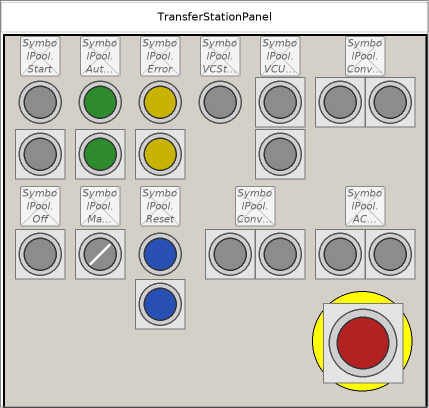
VISUALIZATION V_TransferPanel  // 429x408
VAR_IN_OUT
	Signals : ST_TransferPanel;
END_VAR
    Rectangle (3,34 424x374)
    Ellipse (312,291 100x100)
    PushSwitch (15,129 50x50), tooltip "Activate main contactor", variable: Signals.inputs.PB_ActivateMainContactor, behaviour: TAP, style: Switch-PushSwitch-Gray
    Lamp1 (15,77 50x50), tooltip "Main contactor activeated", variable: Signals.outputs.LED_MainContactorActivated, style: Lamp-Lamp1-Gray
    PushSwitch (75,129 50x50), tooltip "Auto on", variable: Signals.inputs.PB_AutoOn, behaviour: TAP, style: Switch-PushSwitch-Green
    Lamp1 (75,77 50x50), tooltip "Auto activated", variable: Signals.outputs.LED_AutoIsOn, style: Lamp-Lamp1-Green
    Lamp1 (135,77 50x50), tooltip "Error", variable: Signals.outputs.LED_Error, style: Lamp-Lamp1-Yellow
    PushSwitch (135,129 50x50), tooltip "Reset error", variable: Signals.inputs.PB_ErrorReset, behaviour: TAP, style: Switch-PushSwitch-Yellow
    Lamp1 (135,229 50x50), tooltip "Emergency stop", variable: Signals.outputs.LED_EmergencyStop, style: Lamp-Lamp1-Blue
    PushSwitch (135,279 50x50), tooltip "Reset emergency stop", variable: Signals.inputs.PB_EmergencyStopReset, behaviour: TAP, style: Switch-PushSwitch-Blue
    RotarySwitch (75,229 50x50), tooltip "Man/Auto", variable: Signals.inputs.SW_Auto, behaviour: TOGGLE, style: Switch-RotarySwitch-Gray
    Lamp1 (195,77 50x50), tooltip "VC stopped", variable: Signals.outputs.LED_VcStopped, style: Lamp-Lamp1-Gray
    PushSwitch (255,129 50x50), tooltip "VC Down", variable: Signals.inputs.PB_VcDown, behaviour: TAP, style: Switch-PushSwitch-Gray
    PushSwitch (255,77 50x50), tooltip "VC Up", variable: Signals.inputs.PB_VcUp, behaviour: TAP, style: Switch-PushSwitch-Gray
    PushSwitch (365,77 50x50), tooltip "Transfer Conveyor Right", variable: Signals.inputs.PB_Conv_1_Right, behaviour: TAP, style: Switch-PushSwitch-Gray
    PushSwitch (315,77 50x50), tooltip "Transfer Conveyor Left", variable: Signals.inputs.PB_Conv_1_Left, behaviour: TAP, style: Switch-PushSwitch-Gray
    PushSwitch (255,229 50x50), tooltip "VC Conveyor Right", variable: Signals.inputs.PB_VcConvRight, behaviour: TAP, style: Switch-PushSwitch-Gray
    PushSwitch (205,229 50x50), tooltip "VC Conveyor Left", variable: Signals.inputs.PB_VcConvLeft, behaviour: TAP, style: Switch-PushSwitch-Gray
    PushSwitch (365,229 50x50), tooltip "AC Conveyor Right", variable: Signals.inputs.PB_AC_ConvRight, behaviour: TAP, style: Switch-PushSwitch-Gray
    PushSwitch (315,229 50x50), tooltip "AC Conveyor Left", variable: Signals.inputs.PB_AC_ConvLeft, behaviour: TAP, style: Switch-PushSwitch-Gray
    PushSwitch (15,229 50x50), tooltip "Main contactor off", variable: Signals.inputs.PB_MainContactorOff, behaviour: TAP, style: Switch-PushSwitch-Gray
    PushSwitch (323,303 80x80), tooltip "Emergency stop", variable: Signals.inputs.PB_EmergencyStop, behaviour: TOGGLE, style: Switch-PushSwitch-Red
    Image (20,36 40x40), image: SymbolPool.Start
    Image (80,36 40x40), image: SymbolPool.AutoOn
    Image (140,36 40x40), image: SymbolPool.Error
    Image (200,36 40x40), image: SymbolPool.VCStopped
    Image (260,36 40x40), image: SymbolPool.VCUpDown
    Image (345,36 40x40), image: SymbolPool.Conv1_L_R
    Image (235,186 40x40), image: SymbolPool.Conv_L_R
    Image (345,186 40x40), image: SymbolPool.AC_Conv_L_R
    Image (20,186 40x40), image: SymbolPool.Off
    Image (80,186 40x40), image: SymbolPool.ManAuto
    Image (140,186 40x40), image: SymbolPool.Reset
    Textfield (1,2 428x30), "TransferStationPanel"
END_VISUALIZATION

(* stored: Version 1.1.0.1, ProductVersion 3.1.4024.4
   Visu V_TransferPanel: Id {44171979-833f-47b6-84e7-a1f1fe7e7e8b} *)
